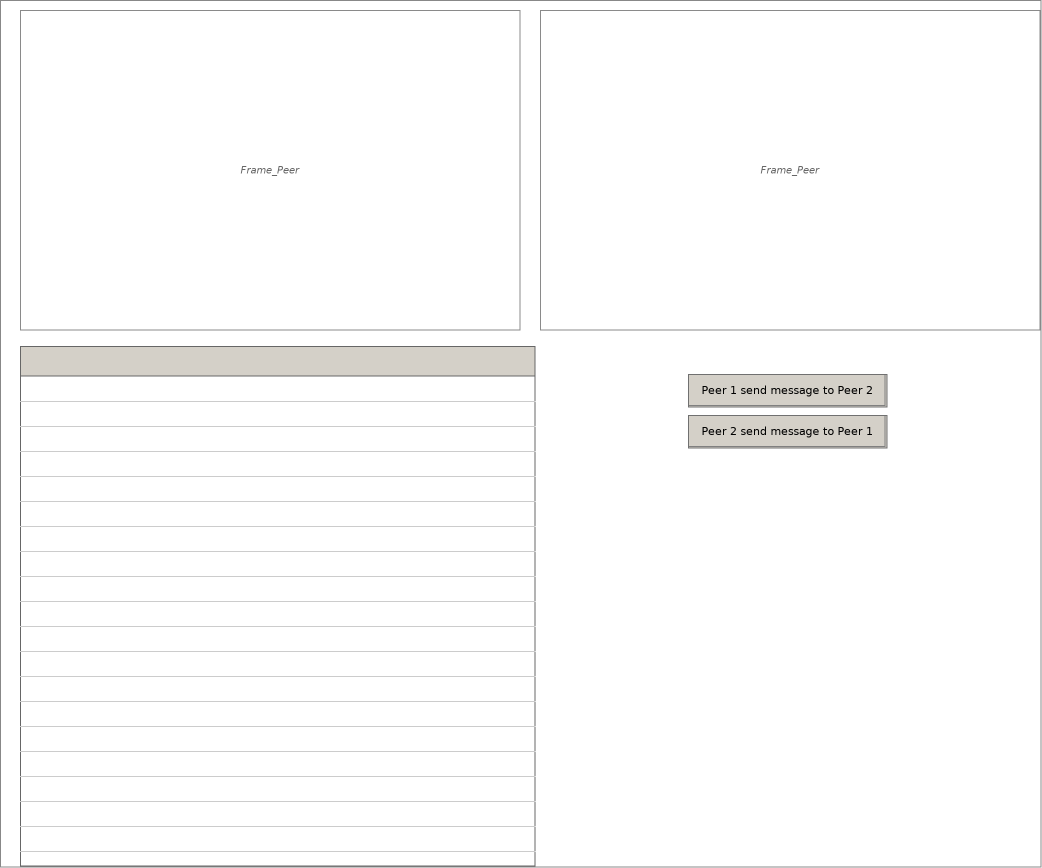
VISUALIZATION VISU_MAIN  // 1042x868
    Frame (20,10 500x320)
        shows Frame_Peer(vio_fbPeer := MAIN.fbDebugPeer1, vio_stMailbox := MAIN.fbDebugPeer1.stMailbox)
    Frame (540,10 500x320)
        shows Frame_Peer(vio_fbPeer := MAIN.fbDebugPeer2, vio_stMailbox := MAIN.fbDebugPeer2.stMailbox)
    Table (20,346 515x520), data array: MAIN.fbMediator.aPeersConnected
        p3854506369: MAIN.fbMediator.aPeersConnected[INDEX].iPeer
        p1892666644: MAIN.fbMediator.aPeersConnected[INDEX].fbMessagesList
        p338671338: MAIN.fbMediator.aPeersConnected[INDEX].nodes
        p2170511999: MAIN.fbMediator.aPeersConnected[INDEX].hList
        p3723444502: MAIN.fbMediator.aPeersConnected[INDEX].nStackPointer
        p1218418051: MAIN.fbMediator.aPeersConnected[INDEX].rMailbox
        p746581629: MAIN.fbMediator.aPeersConnected[INDEX].bMailboxFull
        p3104783080: MAIN.fbMediator.aPeersConnected[INDEX].bMailboxEmpty
        p2237128397: Stack Pointer
        p1757482276: Mailbox Full
        p4088588272: Mailbox Empty
    Button (688,374 199x33), "Peer 1 send message to Peer 2"
        tap MAIN.bPeer1SendMessage
    Button (688,415 199x33), "Peer 2 send message to Peer 1"
        tap MAIN.bPeer2SendMessage
END_VISUALIZATION

(* stored: Version 1.1.0.1, ProductVersion 3.1.4024.0
   Visu VISU_MAIN: Id {dc32d010-e2d9-4283-a62d-29157afbc04b} *)
